// TIA Portal V17 export
// export: Created 2026-04-13T11:12:43.1504213Z, ExportSetting WithDefaults, DisplayName Totally Integrated Automation Portal, DisplayVersion V17 Update 4, DisplayName TIA Portal Openness, DisplayVersion V17 Update 4, DisplayName TIA Portal Version Control Interface, DisplayVersion V17, DisplayName SINAMICS Startdrive Advanced, DisplayVersion V17, DisplayName SINAMICS Startdrive G130, G150, S120, S150, SINAMICS MV, S210, DisplayVersion V17, DisplayName SINAMICS Startdrive G110M, G120, G120C, G120D, G120P, G115D, DisplayVersion V17, DisplayName STEP 7 Professional, DisplayVersion V17 Update 4, DisplayName STEP 7 Safety, DisplayVersion V17, DisplayName WinCC Professional, DisplayVersion V17 Update 4
FUNCTION "相减日期和时间" : Void   // FC3108, STL
TITLE = Data_And_Time减法运算
{ S7_Optimized_Access := 'FALSE' }
VERSION : 0.1
// stored: AutoNumber true, UDAEnableTagReadback false
   VAR_INPUT
      被减时间 : Pointer;   // 被减时间(Data_And_Time类型)
      减数时间 : Pointer;   // 减数(Data_And_Time类型)
      TimeOver : Bool;   // 时间到达
   END_VAR
   VAR_OUTPUT
      剩余时间 : Pointer;   // 剩余时间(Data_And_Time类型)
   END_VAR
   VAR_TEMP
      Minu : Struct
         year : Int;   // 年
         mouth : Int;   // 月
         day : Int;   // 日
         hour : Int;   // 时
         min : Int;   // 分
         sec : Int;   // 秒
      END_STRUCT;
      Sub : Struct
         year : Int;   // 年
         mouth : Int;   // 月
         day : Int;   // 日
         hour : Int;   // 时
         min : Int;   // 分
         sec : Int;   // 秒
      END_STRUCT;
      Res : Struct
         year : Int;   // 年
         mouth : Int;   // 月
         day : Int;   // 日
         hour : Int;   // 时
         min : Int;   // 分
         sec : Int;   // 秒
      END_STRUCT;
      MinuDB : Int;
      SubDB : Int;
      ResDB : Int;
      temp1 : Byte;
      temp2 : Byte;
      temp3 : Byte;
      temp4 : Byte;
      temp5 : Byte;
      temp6 : Byte;
      temp7 : Byte;
      temp8 : Byte;
      temp9 : Byte;
      temp10 : Byte;
      temp11 : Byte;
      temp12 : Byte;
      temp13 : Byte;
      temp14 : Byte;
      temp15 : Byte;
      temp16 : Byte;
   END_VAR
BEGIN

NETWORK
TITLE = 指针提取
      L     P##被减时间;  //提取被减时间
      LAR1;
      L     P##减数时间;  //提取被时间
      LAR2;

      L     W [AR1, P#0.0];
      T     #MinuDB;
      L     W [AR2, P#0.0];
      T     #SubDB;
      L     W [AR1, P#4.0];
      LAR1;
      L     W [AR2, P#4.0];
      LAR2;

      A     #TimeOver;
      JC    OVER;


NETWORK
TITLE = 被减时间提取，转化为DEC
      OPN   DB [#MinuDB];
      L     DBB [AR1, P#0.0];
      SRW   4;
      L     10;
      *I;
      T     #temp1;
      L     DBB [AR1, P#0.0];
      L     b#16#0f;
      AW;
      L     #temp1;
      +I;
      T     #Minu.year;  // year

      OPN   DB [#MinuDB];
      L     DBB [AR1, P#1.0];
      SRW   4;
      L     10;
      *I;
      T     #temp2;
      L     DBB [AR1, P#1.0];
      L     b#16#0f;
      AW;
      L     #temp2;
      +I;
      T     #Minu.mouth;  // mouth

      OPN   DB [#MinuDB];
      L     DBB [AR1, P#2.0];
      SRW   4;
      L     10;
      *I;
      T     #temp3;
      L     DBB [AR1, P#2.0];
      L     b#16#0f;
      AW;
      L     #temp3;
      +I;
      T     #Minu.day;  // day

      OPN   DB [#MinuDB];
      L     DBB [AR1, P#3.0];
      SRW   4;
      L     10;
      *I;
      T     #temp4;
      L     DBB [AR1, P#3.0];
      L     b#16#0f;
      AW;
      L     #temp4;
      +I;
      T     #Minu.hour;  // hour

      OPN   DB [#MinuDB];
      L     DBB [AR1, P#4.0];
      SRW   4;
      L     10;
      *I;
      T     #temp5;
      L     DBB [AR1, P#4.0];
      L     b#16#0f;
      AW;
      L     #temp5;
      +I;
      T     #Minu.min;  // min

      OPN   DB [#MinuDB];
      L     DBB [AR1, P#5.0];
      SRW   4;
      L     10;
      *I;
      T     #temp6;
      L     DBB [AR1, P#5.0];
      L     b#16#0f;
      AW;
      L     #temp6;
      +I;
      T     #Minu.sec;  // sec


NETWORK
TITLE = 减时间提取，转化为DEC
      OPN   DB [#SubDB];
      L     DBB [AR2, P#0.0];
      SRW   4;
      L     10;
      *I;
      T     #temp7;
      L     DBB [AR2, P#0.0];
      L     b#16#0f;
      AW;
      L     #temp7;
      +I;
      T     #Sub.year;  // year

      OPN   DB [#SubDB];
      L     DBB [AR2, P#1.0];
      SRW   4;
      L     10;
      *I;
      T     #temp8;
      L     DBB [AR2, P#1.0];
      L     b#16#0f;
      AW;
      L     #temp8;
      +I;
      T     #Sub.mouth;  // mouth

      OPN   DB [#SubDB];
      L     DBB [AR2, P#2.0];
      SRW   4;
      L     10;
      *I;
      T     #temp9;
      L     DBB [AR2, P#2.0];
      L     b#16#0f;
      AW;
      L     #temp9;
      +I;
      T     #Sub.day;  // day

      OPN   DB [#SubDB];
      L     DBB [AR2, P#3.0];
      SRW   4;
      L     10;
      *I;
      T     #temp10;
      L     DBB [AR2, P#3.0];
      L     b#16#0f;
      AW;
      L     #temp10;
      +I;
      T     #Sub.hour;  // hour

      OPN   DB [#SubDB];
      L     DBB [AR2, P#4.0];
      SRW   4;
      L     10;
      *I;
      T     #temp11;
      L     DBB [AR2, P#4.0];
      L     b#16#0f;
      AW;
      L     #temp11;
      +I;
      T     #Sub.min;  // min

      OPN   DB [#SubDB];
      L     DBB [AR2, P#5.0];
      SRW   4;
      L     10;
      *I;
      T     #temp12;
      L     DBB [AR2, P#5.0];
      L     b#16#0f;
      AW;
      L     #temp12;
      +I;
      T     #Sub.sec;  // sec


NETWORK
TITLE = 减法运算
      L     #Minu.year;
      L     #Sub.year;
      -I;
      T     #Res.year;

      L     #Minu.mouth;
      L     #Sub.mouth;
      -I;
      T     #Res.mouth;

      L     #Minu.day;
      L     #Sub.day;
      -I;
      T     #Res.day;

      L     #Minu.hour;
      L     #Sub.hour;
      -I;
      T     #Res.hour;

      L     #Minu.min;
      L     #Sub.min;
      -I;
      T     #Res.min;

      L     #Minu.sec;
      L     #Sub.sec;
      -I;
      T     #Res.sec;


NETWORK
TITLE = 被减数小于减数，向高位借1
      A(;
      L     #Res.sec;
      L     0;
      <I;
      );
      JCN   _001;
      L     #Res.sec;
      L     60;
      +I;
      T     #Res.sec;
      L     #Res.min;
      L     1;
      -I;
      T     #Res.min;
_001: A(;
      L     #Res.min;
      L     0;
      <I;
      );
      JCN   _002;
      L     #Res.min;
      L     60;
      +I;
      T     #Res.min;
      L     #Res.hour;
      L     1;
      -I;
      T     #Res.hour;
_002: A(;
      L     #Res.hour;
      L     0;
      <I;
      );
      JCN   _003;
      L     #Res.hour;
      L     24;
      +I;
      T     #Res.hour;
      L     #Res.day;
      L     1;
      -I;
      T     #Res.day;
_003: A(;
      L     #Res.day;
      L     0;
      <I;
      );
      JCN   _004;
      L     #Res.day;
      L     30;
      +I;
      T     #Res.day;
      L     #Res.mouth;
      L     1;
      -I;
      T     #Res.mouth;
_004: A(;
      L     #Res.mouth;
      L     0;
      <I;
      );
      JCN   _111;
      L     #Res.mouth;
      L     12;
      +I;
      T     #Res.mouth;
      L     #Res.year;
      L     1;
      -I;
      T     #Res.year;
_111: NOP   0;
      JU    Resi;

NETWORK
TITLE = time over
OVER: L     0;
      T     #Res.year;
      T     #Res.mouth;
      T     #Res.day;
      T     #Res.hour;
      T     #Res.min;
      T     #Res.sec;


NETWORK
TITLE = 差值赋值到剩余时间
Resi: L     P##剩余时间;  //提取剩余时间
      LAR1;
      L     W [AR1, P#0.0];
      T     #ResDB;
      L     W [AR1, P#4.0];
      LAR1;

      OPN   DB [#ResDB];
      L     #Res.year;
      T     DBB [AR1, P#0.0];
      L     #Res.mouth;
      T     DBB [AR1, P#1.0];
      L     #Res.day;
      T     DBB [AR1, P#2.0];
      L     #Res.hour;
      T     DBB [AR1, P#3.0];
      L     #Res.min;
      T     DBB [AR1, P#4.0];
      L     #Res.sec;
      T     DBB [AR1, P#5.0];



NETWORK
TITLE = RLO
      SET;
      SAVE;

END_FUNCTION
